// TIA Portal V20 export
TYPE "zm_MachineStatus"
// stored: Access Published
   STRUCT
      Aborted : Bool;
      Stopped : Bool;
      Idle : Bool;
      Execute : Bool;
      Held : Bool;
      Suspended : Bool;
      Complete : Bool;
   END_STRUCT;
END_TYPE
